# EPICS autosave request: CAENV895/iocBoot/iocCAENV895-IOC-01/auto_settings.req
file configMenu_settings.req P=$(P),CONFIG=vmeconfig
